(* PLC project Generated.project, CODESYS CODESYS V3.5 SP19 Patch 1 *)
(* stored: creationDateTime 2026-09-06T13:00:42.436101, modificationDateTime 2026-09-06T13:00:42.436101 *)

(* ======================================================================= 🪜 ST_SpeedStepTable — Table des paliers de vitesse contacteurs ─────────────────────────────────────────────────────────────── 🎯 Rôle : Structure de configuration des contacteurs et seuils par palier 📄 Doc métier : DOC/AF/AF_Partie-10_Fonction_Winch_v2.1.md ======================================================================= *)
TYPE ST_SpeedStepTable : STRUCT
  P1R1 : BOOL;  (* === PALIER 1 (VITESSE MINIMALE) === Contacteur 1 pour Palier 1 *)
  P1R2 : BOOL;  (* Contacteur 2 pour Palier 1 *)
  P1R3 : BOOL;  (* Contacteur 3 pour Palier 1 *)
  P1R4 : BOOL;  (* Contacteur 4 pour Palier 1 *)
  P2R1 : BOOL;  (* === PALIER 2 === Contacteur 1 pour Palier 2 *)
  P2R2 : BOOL;  (* Contacteur 2 pour Palier 2 *)
  P2R3 : BOOL;  (* Contacteur 3 pour Palier 2 *)
  P2R4 : BOOL;  (* Contacteur 4 pour Palier 2 *)
  P3R1 : BOOL;  (* === PALIER 3 === Contacteur 1 pour Palier 3 *)
  P3R2 : BOOL;  (* Contacteur 2 pour Palier 3 *)
  P3R3 : BOOL;  (* Contacteur 3 pour Palier 3 *)
  P3R4 : BOOL;  (* Contacteur 4 pour Palier 3 *)
  P4R1 : BOOL;  (* === PALIER 4 === Contacteur 1 pour Palier 4 *)
  P4R2 : BOOL;  (* Contacteur 2 pour Palier 4 *)
  P4R3 : BOOL;  (* Contacteur 3 pour Palier 4 *)
  P4R4 : BOOL;  (* Contacteur 4 pour Palier 4 *)
  P5R1 : BOOL;  (* === PALIER 5 (VITESSE MAXIMALE) === Contacteur 1 pour Palier 5 *)
  P5R2 : BOOL;  (* Contacteur 2 pour Palier 5 *)
  P5R3 : BOOL;  (* Contacteur 3 pour Palier 5 *)
  P5R4 : BOOL;  (* Contacteur 4 pour Palier 5 *)
  StepThreshold_Pct : ARRAY[1..5] OF REAL;  (* === SEUILS DE TRANSITION (%) === Seuils de changement de palier (0..100%) *)
END_STRUCT;
END_TYPE
